{attribute 'qualified_only'}
{attribute 'strict'}
TYPE E_LSS_State :
(
	//GENERIC
	ABORTED				,
	READY				,
	//MANUAL_MODE			:=50, /manual mode not needed.
	ERROR				,
	//SPECIFIC FOR EVERY STATION
	TRIGGER				,
	MEASUREMENT			,
	DONE				,
	RESULTS				,
	RESET_CMD			,
	HOMING				,
	MANUAL_MODE			
);
END_TYPE

(* stored: Version 1.1.0.1, ProductVersion 3.1.4026.18
   DUT E_LSS_State: Id {5ddfb4d9-7fc1-463c-94a3-7a2a15a0ec39} *)
